PROGRAM PRG_Lab
VAR
	fbStatusLight : FB_StatusLight;
	
	fbSeparator : FB_Separator;
	
	fbRFID : FB_RFID;
	
	fbConveyor : FB_Conveyor;
	
	fbFillLevel1 : FB_FillLevel;
	fbFillLevel2 : FB_FillLevel;
	fbFillLevel3 : FB_FillLevel;
	
	fbDisp1 : FB_Dispenser;
	fbDisp2 : FB_Dispenser;
	fbDisp3 : FB_Dispenser;
	
	fbManX  : FB_ManipulatorAxis;
	fbManY  : FB_ManipulatorAxis;
	fbManZ  : FB_ManipulatorAxis;
	fbManGrip 	: FB_ManipulatorAxis;
	
	fbWaage : FB_Waage;
	
	fbHeating : FB_HeatingSystem;
	
	nState : INT := 0;
	nCount : INT := 0;
	
	timer : TON;
END_VAR

fbStatusLight(
	bRed=> IFC_HW.AmpelRot,
	bYellow=> IFC_HW.AmpelGelb,
	bGreen=> IFC_HW.AmpelGrun);

fbSeparator(
	bSensor1:= IFC_HW.EinzelSens1, 
	bSensor2:= IFC_HW.EinzelSens2, 
	bR1AKT1=> IFC_HW.R1AKT1, 
	bR1AKT2=> IFC_HW.R1AKT2,
	bR2AKT1=> IFC_HW.R2AKT1, 
	bR2AKT2=> IFC_HW.R2AKT2,
	bNoBottle=> IFC_HW.NoBottle,	
	bWrongBottle=> IFC_HW.WrongBottle);
	
fbRFID( 
	sSeriennummer=> IFC_HW.IdNachricht);

fbConveyor(
	ax:= IFC_HW.BandMotor);

fbFillLevel1(
	nLevelIn:= IFC_HW.FillSens1,
	nMaxLevel:= IFC_HW.MaxFillLevel,
	nLevelPercent=> IFC_HW.FillLevelPercent1,
	nLevelGramm=> IFC_HW.FillLevelGramm1);
fbFillLevel2(
	nLevelIn:= IFC_HW.FillSens2,
	nMaxLevel:= IFC_HW.MaxFillLevel,
	nLevelPercent=> IFC_HW.FillLevelPercent2,
	nLevelGramm=> IFC_HW.FillLevelGramm2);
fbFillLevel3(
	nLevelIn:= IFC_HW.FillSens3,
	nMaxLevel:= IFC_HW.MaxFillLevel,
	nLevelPercent=> IFC_HW.FillLevelPercent3,
	nLevelGramm=> IFC_HW.FillLevelGramm3);
	
fbDisp1(
	ax:= IFC_HW.BandExtruder1);
fbDisp2(
	ax:= IFC_HW.BandExtruder2);
fbDisp3(
	ax:= IFC_HW.BandExtruder3);

fbManX(
	aAchse:= IFC_HW.ManAchseX,
	bEndSchalterMin:=IFC_HW.ManEndX,
	bEndSchalterMax:=IFC_HW.ManEndX2);
fbManY(
	aAchse:= IFC_HW.ManAchseY,
	bEndSchalterMin:=IFC_HW.ManEndY,
	bEndSchalterMax:=IFC_HW.ManEndY2);
fbManZ(
	aAchse:= IFC_HW.ManAchseZ,
	bEndSchalterMin:=IFC_HW.ManEndZ,
	bEndSchalterMax:=IFC_HW.ManEndZ2);
	
fbManGrip(
	aAchse:= IFC_HW.ManAchseGrip,
	bEndSchalterMin:=IFC_HW.ManEndGrip,
	bEndSchalterMax:=IFC_HW.ManEndGrip2);
	
fbWaage(
	bNullsetzen:= IFC_HW.WaageNull,
	iMesswert=> IFC_HW.WaageMesswert);
	
fbHeating(
	nMaxTemp:= IFC_HW.MaxTemp,
	nTemp:= (IFC_HW.TempSens1 + IFC_HW.TempSens2)/2,
	bVentilator1=> IFC_HW.Ventilator1,
	bVentilator2=> IFC_HW.Ventilator2,
	bVentilator3=> IFC_HW.Ventilator3,
	nHeizpatrone=> IFC_HW.Heizpatrone);	
	
CASE nState OF
0: // Off
	fbStatusLight.eStatus := State.Off;
	fbSeparator.bEnable := FALSE;
	fbConveyor.bEnable := FALSE;
	fbDisp1.bEnable := FALSE;
	fbDisp2.bEnable := FALSE;
	fbDisp3.bEnable := FALSE;
	fbHeating.bEnable := FALSE;
	fbManX.bEnable := FALSE;
	fbManY.bEnable := FALSE;
	fbManZ.bEnable := FALSE;
	fbManGrip.bEnable := FALSE;
	
	nState := nState + 1;
	
1: // Turn on
	fbStatusLight.eStatus := State.Busy;
	fbSeparator.bEnable := TRUE;
	fbConveyor.bEnable := TRUE;
	fbDisp1.bEnable := TRUE;
	fbDisp2.bEnable := TRUE;
	fbDisp3.bEnable := TRUE;
	fbHeating.bEnable := TRUE;
	IFC_HW.Brake := TRUE;
	fbManZ.bEnable := TRUE;
	IF fbManZ.eOutState = State.Ready THEN
		IFC_HW.Brake := FALSE;
		fbManX.bEnable := TRUE;
		fbManY.bEnable := TRUE;
		fbManGrip.bEnable := TRUE;
	END_IF
	
	IF fbSeparator.eStatus = State.Ready
		AND fbConveyor.eStatus = State.Ready
		AND fbDisp1.eStatus = State.Ready
		AND fbDisp2.eStatus = State.Ready
		AND fbDisp3.eStatus = State.Ready
		AND fbHeating.eStatus = State.Ready
		AND fbManX.eOutState = State.Ready
		AND fbManY.eOutState = State.Ready
		AND fbManGrip.eOutState = State.Ready THEN
		nState := nState + 1;
	END_IF

2: // check error
	IF nCount >= 4 THEN
		fbStatusLight.eStatus := State.Error;
		IFC_HW.StorageFull := TRUE;
		IF GVL_SAFETY.safeOverruled AND GVL_SAFETY.bAcknowledge_Button THEN
			IFC_HW.StorageFull := FALSE;
			GVL_SAFETY.safeOverruled := FALSE;
			nCount := 0;
			nState := nState + 1;
		END_IF
	ELSIF  NOT IFC_HW.EinzelSens2 AND NOT IFC_HW.EinzelSens3 THEN
		fbStatusLight.eStatus := State.Error;
		IFC_HW.NoBottle := TRUE;
		IF GVL_SAFETY.bAcknowledge_Button THEN
			IFC_HW.NoBottle := FALSE;
			nState := 1;
		END_IF
	ELSIF (NOT IFC_HW.EinzelSens2 AND IFC_HW.EinzelSens3) OR (IFC_HW.EinzelSens2 AND IFC_HW.EinzelSens3)THEN
		fbStatusLight.eStatus := State.Error;
		IFC_HW.WrongBottle := TRUE;
		IF GVL_SAFETY.bAcknowledge_Button THEN
			IFC_HW.WrongBottle := FALSE;
			nState := 1;
		END_IF
	ELSIF IFC_HW.FillLevelPercent1 < 5 OR IFC_HW.FillLevelPercent2 < 5 OR IFC_HW.FillLevelPercent3 < 5 THEN
		fbStatusLight.eStatus := State.Error;
		IFC_HW.GranulateEmpty := TRUE;
		IF GVL_SAFETY.bAcknowledge_Button THEN
			IFC_HW.GranulateEmpty := FALSE;
			nState := 1;
		END_IF
	ELSE
		nState := nState + 1;
	END_IF
	
3: // All systems ready
	fbStatusLight.eStatus := State.Ready;
	
	IF (GVL_SAFETY.bBetrieb_Button OR GVL_VIS.bStartFactoryHMI) AND NOT GVL_SAFETY.safeOverruled THEN
		GVL_SAFETY.bBetrieb_Button := FALSE; // reset
		nState := nState + 1;
	END_IF
	
4: // read RFID
	fbStatusLight.eStatus := State.Busy;
	//fbRFID.bSensorTrager := TRUE;
	
	//IF fbRFID.bFertig THEN
		//fbRFID.bSensorTrager := FALSE;
		nState := nState + 1;
	//END_IF
	
5: // separate container
	fbSeparator.bExecute := TRUE;
	
	IF fbSeparator.eStatus = State.Done THEN
		fbSeparator.bExecute := FALSE;
		nState := nState + 1;
	END_IF
	
6: // turn on conveyor and wait for container to arrive at BandSens1
	fbConveyor.eDirection := MC_Direction.MC_Positive_Direction;
	fbConveyor.nVel := 40;
	fbConveyor.bExecute := TRUE;
	
	IF IFC_HW.BandSens1 THEN
		timer(IN := TRUE, PT := T#500MS);
		IF timer.Q THEN
			fbConveyor.bExecute := FALSE;
			timer(IN := FALSE);
			nState := nState + 1;
		END_IF
	END_IF
	
7: // fill container from first dispenser
	fbDisp1.nDispenseGrams := IFC_HW.BandFullmenge1;
	fbDisp1.bExecute := TRUE;
	
	IF fbDisp1.eStatus = State.Done THEN
		fbDisp1.bExecute := FALSE;
		nState := nState + 1;
	END_IF
	
8: // continue conveyor to second dispenser (BandSens2)
	fbConveyor.eDirection := MC_Direction.MC_Positive_Direction;
	fbConveyor.nVel := 40;
	
	fbConveyor.bExecute := TRUE;
	
	IFC_HW.BandHub1 := TRUE;
	
	IF IFC_HW.BandSens2 THEN
		timer(IN := TRUE, PT := T#500MS);
		IF timer.Q THEN
			fbConveyor.bExecute := FALSE;
			IFC_HW.BandHub1 := FALSE;
			timer(IN := FALSE);
			nState := nState + 1;
		END_IF
	END_IF
	
9: // fill container from second dispenser
	fbDisp2.nDispenseGrams := IFC_HW.BandFullmenge2;
	fbDisp2.bExecute := TRUE;
	
	IF fbDisp2.eStatus = State.Done THEN
		fbDisp2.bExecute := FALSE;
		nState := nState + 1;
	END_IF
	
10: // continue conveyor to third dispenser (BandSens3)
	fbConveyor.eDirection := MC_Direction.MC_Positive_Direction;
	fbConveyor.nVel := 40;
	fbConveyor.bExecute := TRUE;
	
	IFC_HW.BandHub2 := TRUE;
	
	IF IFC_HW.BandSens3 THEN
		timer(IN := TRUE, PT := T#500MS);
		IF timer.Q THEN
			fbConveyor.bExecute := FALSE;
			IFC_HW.BandHub2 := FALSE;
			timer(IN := FALSE);
			nState := nState + 1;
		END_IF
	END_IF
	
11: // fill container from second dispenser
	fbDisp3.nDispenseGrams := IFC_HW.BandFullmenge3;
	fbDisp3.bExecute := TRUE;
	
	IF fbDisp3.eStatus = State.Done THEN
		fbDisp3.bExecute := FALSE;
		nState := nState + 1;
	END_IF
	
12: // continue conveyor to end of line (BandSens4)
	fbConveyor.eDirection := MC_Direction.MC_Positive_Direction;
	fbConveyor.nVel := 40;
	fbConveyor.bExecute := TRUE;
	
	IFC_HW.BandHub3 := TRUE;
	
	IF IFC_HW.BandSens4 THEN
		timer(IN := TRUE, PT := T#500MS);
		IF timer.Q THEN
			fbConveyor.bExecute := FALSE;
			IFC_HW.BandHub3 := FALSE;
			timer(IN := FALSE);
			nState := nState + 1;
		END_IF
	END_IF

13: // open Gripper
	fbManGrip.fVelocity := 3;	
	fbManGrip.fPosition := 6;
	
	fbManGrip.bExecute := TRUE;	
	
	IF fbManGrip.eOutState = State.Done THEN
		fbManGrip.bExecute := FALSE;
		nState := nState + 1;
	END_IF
		
14: // goto container x, y
	fbManX.fVelocity := 30;
	fbManY.fVelocity := 30;
	
	fbManX.fPosition := 31;
	fbManY.fPosition := 145;
	
	fbManX.bExecute := TRUE;
	fbManY.bExecute := TRUE;
	
	IF fbManX.eOutState = State.Done AND fbManY.eOutState = State.Done THEN
		fbManX.bExecute := FALSE;
		fbManY.bExecute := FALSE;
		nState := nState + 1;
	END_IF
	
15: // goto container z	
	fbManZ.fVelocity := 30;
	
	fbManZ.fPosition := 132;
	
	IFC_HW.Brake := TRUE;
	fbManZ.bExecute := TRUE;
	
	IF fbManZ.eOutState = State.Done THEN
		fbManZ.bExecute := FALSE;
		IFC_HW.Brake := FALSE;
		nState := nState + 1;
	END_IF

16: // close Gripper
	fbManGrip.fPosition := 8.5;
	
	fbManGrip.bExecute := TRUE;	
	
	IF fbManGrip.eOutState = State.Done THEN
		fbManGrip.bExecute := FALSE;
		nState := nState + 1;
	END_IF

17: // move Z UP
	fbManZ.fPosition := 70;

	IFC_HW.Brake := TRUE;
	fbManZ.bExecute := TRUE;	
	
	IF fbManZ.eOutState = State.Done THEN
		fbManZ.bExecute := FALSE;
		IFC_HW.Brake := FALSE;
		nState := nState + 1;
	END_IF

18: // goto scale x, y
	fbManX.fPosition := 37;
	fbManY.fPosition := 7;
	
	fbManX.bExecute := TRUE;
	fbManY.bExecute := TRUE;
	
	IF fbManX.eOutState = State.Done AND fbManY.eOutState = State.Done THEN
		fbManX.bExecute := FALSE;
		fbManY.bExecute := FALSE;
		nState := nState + 1;
	END_IF

19: // set scale to zero	
	//IFC_HW.WaageNull := TRUE;
	
	//IF fBWaage.iMesswert = 0 THEN
		nState := nState + 1;
	//END_IF

20: // goto scale z	
	fbManZ.fPosition := 132.5;
	
	IFC_HW.Brake := TRUE;
	fbManZ.bExecute := TRUE;
	
	IF fbManZ.eOutState = State.Done THEN
		fbManZ.bExecute := FALSE;
		IFC_HW.Brake := FALSE;
		nState := nState + 1;
	END_IF
	
21: // open Gripper		
	fbManGrip.fPosition := 6;
	
	fbManGrip.bExecute := TRUE;
	
	IF fbManGrip.eOutState = State.Done THEN
		fbManGrip.bExecute := FALSE;
		nState := nState + 1;
	END_IF
	
22: // scale 
	nState := nState + 1;
	
23: // close Gripper
	fbManGrip.fPosition := 8.5;	
	
	fbManGrip.bExecute := TRUE;	
	
	IF fbManGrip.eOutState = State.Done THEN
		fbManGrip.bExecute := FALSE;
		nState := nState + 1;
	END_IF

24: // move Z UP	
	fbManZ.fPosition := 70;
	
	IFC_HW.Brake := TRUE;
	fbManZ.bExecute := TRUE;
	
	IF fbManZ.eOutState = State.Done THEN
		fbManZ.bExecute := FALSE;
		IFC_HW.Brake := FALSE;
		nState := nState + 1;
	END_IF
	
25: // goto heating x, y
	fbManX.fPosition := 220.5;
	fbManY.fPosition := 6;
	
	fbManX.bExecute := TRUE;
	fbManY.bExecute := TRUE;
	
	IF fbManX.eOutState = State.Done AND fbManY.eOutState = State.Done THEN
		fbManX.bExecute := FALSE;
		fbManY.bExecute := FALSE;
		nState := nState + 1;
	END_IF

26: // goto heating z	
	fbManZ.fPosition := 180;
	
	IFC_HW.Brake := TRUE;
	fbManZ.bExecute := TRUE;
	
	IF fbManZ.eOutState = State.Done THEN
		fbManZ.bExecute := FALSE;
		IFC_HW.Brake := FALSE;
		nState := nState + 1;
	END_IF

27: // open Gripper	
	fbManGrip.fPosition := 6;
	
	fbManGrip.bExecute := TRUE;	
	
	IF fbManGrip.eOutState = State.Done THEN
		fbManGrip.bExecute := FALSE;
		nState := nState + 1;
	END_IF
	
28: // heating 
	fbHeating.bExecute := TRUE;
	
	IF fbHeating.eStatus = State.Done THEN
		fbHeating.bExecute := FALSE;
		nState := nState + 1;
	END_IF

29: // close Gripper
	fbManGrip.fPosition := 8.5;	
	
	fbManGrip.bExecute := TRUE;	
	
	IF fbManGrip.eOutState = State.Done THEN
		fbManGrip.bExecute := FALSE;
		nState := nState + 1;
	END_IF

30: // move Z UP	
	fbManZ.fPosition := 70;
	
	IFC_HW.Brake := TRUE;
	fbManZ.bExecute := TRUE;
	
	IF fbManZ.eOutState = State.Done THEN
		fbManZ.bExecute := FALSE;
		IFC_HW.Brake := FALSE;
		nState := nState + 1;
	END_IF

31: // goto storage x, y
	CASE nCount OF		
	0: // storage 1
		fbManX.fPosition := 110.5;
	1: // storage 2
		fbManX.fPosition := 161.5;
	2: // storage 3
		fbManX.fPosition := 212.5;
	3: // storage 4
		fbManX.fPosition := 263;	
	END_CASE
	
	fbManY.fPosition := 138;
	
	fbManX.bExecute := TRUE;
	fbManY.bExecute := TRUE;
	
	IF fbManX.eOutState = State.Done AND fbManY.eOutState = State.Done THEN
		fbManX.bExecute := FALSE;
		fbManY.bExecute := FALSE;
		nCount := nCount + 1;
		nState := nState + 1;
	END_IF

32: // goto storage z	
	fbManZ.fPosition := 128;
	
	IFC_HW.Brake := TRUE;
	fbManZ.bExecute := TRUE;
	
	IF fbManZ.eOutState = State.Done THEN
		fbManZ.bExecute := FALSE;
		IFC_HW.Brake := FALSE;
		nState := nState + 1;
	END_IF	
	
33: // open Gripper		
	fbManGrip.fPosition := 6;
	
	fbManGrip.bExecute := TRUE;
	
	IF fbManGrip.eOutState = State.Done THEN
		fbManGrip.bExecute := FALSE;
		nState := nState + 1;
	END_IF
	
34: // move Z UP
	fbManZ.fPosition := 80;
	
	IFC_HW.Brake := TRUE;
	fbManZ.bExecute := TRUE;
	
	IF fbManZ.eOutState = State.Done THEN
		fbManZ.bExecute := FALSE;
		IFC_HW.Brake := FALSE;
		nState := nState + 1;
	END_IF
	
35: // goto container x, y
	fbManX.fPosition := 31;
	fbManY.fPosition := 145;
	
	fbManX.bExecute := TRUE;
	fbManY.bExecute := TRUE;
	
	IF fbManX.eOutState = State.Done AND fbManY.eOutState = State.Done THEN
		fbManX.bExecute := FALSE;
		fbManY.bExecute := FALSE;
		nState := nState + 1;
	END_IF
	
36: // Done
	fbStatusLight.eStatus := State.Done;
	
	timer(IN := TRUE, PT := T#3000MS);
	
	IF timer.Q THEN
		timer(IN := FALSE);
		nState := 1;
	END_IF
	
END_CASE

END_PROGRAM

(* stored: Version 1.1.0.1, ProductVersion 3.1.4024.11
   POU PRG_Lab: Id {56de3c86-00a0-4a8b-ae04-45bb1f6f07de}, SpecialFunc None *)
